// TIA Portal V17 export
// export: Created 2025-06-26T06:49:21.3068873Z, ExportSetting WithDefaults, DisplayName Totally Integrated Automation Portal, DisplayVersion V17 Update 8, DisplayName TIA Portal Openness, DisplayVersion V17 Update 8, DisplayName TIA Portal Version Control Interface, DisplayVersion V17, DisplayName STEP 7 Professional, DisplayVersion V17 Update 8, DisplayName STEP 7 Safety, DisplayVersion V17 Update 6, DisplayName WinCC Advanced, DisplayVersion V17 Update 8
DATA_BLOCK "RDREC_GetDiagInfo"   // DB17
// stored: AutoNumber true, DBAccessibleFromOPCUA true, InstanceOfName RDREC_SFB, OfSystemLibElement RDREC, OfSystemLibVersion 1.0
"RDREC_SFB"
   // VAR_INPUT
   //    REQ : Bool;
   //    ID : HW_IO;
   //    INDEX : DInt;
   //    MLEN : UInt;
   // END_VAR
   // VAR_OUTPUT
   //    VALID : Bool;
   //    BUSY : Bool;
   //    ERROR : Bool;
   //    STATUS : DWord;
   //    LEN : UInt;
   // END_VAR
   // VAR_IN_OUT
   //    RECORD : Variant;
   // END_VAR
BEGIN
END_DATA_BLOCK
